KUKA KRL data list: calc_positions.dat

&ACCESS RV1
&PARAM EDITMASK = *
&PARAM TEMPLATE = C:\KRC\Roboter\Template\ExpertVorgabe
DEFDAT calc_positions PUBLIC

ENDDAT
